FUNCTION_BLOCK PUBLIC FB_SocketOnCommand IMPLEMENTS I_Command
VAR
	refSocket : REFERENCE TO FB_Socket;
END_VAR

METHOD Execute
IF (__ISVALIDREF(THIS^.refSocket)) THEN
	THIS^.refSocket.On();
END_IF
END_METHOD

METHOD FB_init : BOOL
VAR_INPUT
	bInitRetains : BOOL; // if TRUE, the retain variables are initialized (warm start / cold start)
	bInCopyCode : BOOL;  // if TRUE, the instance afterwards gets moved into the copy code (online change)
	refNewSocket : REFERENCE TO FB_Socket;
END_VAR
IF (__ISVALIDREF(refNewSocket)) THEN
	THIS^.refSocket REF= refNewSocket;
ELSE
	THIS^.refSocket REF= 0;
END_IF
END_METHOD

METHOD Undo
IF (__ISVALIDREF(THIS^.refSocket)) THEN
	THIS^.refSocket.Off();
END_IF
END_METHOD

END_FUNCTION_BLOCK

(* stored: Version 1.1.0.1, ProductVersion 3.1.4020.3
   POU FB_SocketOnCommand: Id {eb2e5cd4-b6f9-41c2-bfb5-fea646599ebe}, SpecialFunc None
   Method Execute: Id {00744c42-2535-4c07-9d72-9dfd58f4279b}
   Method FB_init: Id {b23704c1-7621-4b32-8be0-30a679a8c783}
   Method Undo: Id {0f1590db-7995-473d-af6f-20187b5a3c44} *)
